# EPICS substitutions: epics-loctite-eqcl25App/Db/ledData.substitutions
file "${TOP}/loctite-chx-ledApp/Db/ledData.db"
{
pattern
{PREFIX, CHNM, RINTENADDR, WINTENADDR, SELSTATADDR, SELADDR, TEMPADDR, RTIMEADDR, WTIMEADDR}
{"$(PREFIX)", "{LOCTITE:Chan1}", 5104, 7104, 5100, 7100, 5070, 5105, 7105}
{"$(PREFIX)", "{LOCTITE:Chan2}", 5106, 7106, 5101, 7101, 5071, 5107, 7107}
{"$(PREFIX)", "{LOCTITE:Chan3}", 5108, 7108, 5102, 7102, 5072, 5109, 7109}
{"$(PREFIX)", "{LOCTITE:Chan4}", 5110, 7110, 5103, 7103, 5073, 5111, 7111}
}
